// TIA Portal V17 export
// export: Created 2023-06-23T18:33:41.3605252Z, ExportSetting WithDefaults, DisplayName Totally Integrated Automation Portal, DisplayVersion V17, DisplayName TIA Portal Openness, DisplayVersion V17, DisplayName TIA Portal Version Control Interface, DisplayVersion V17, DisplayName STEP 7 Professional, DisplayVersion V17, DisplayName STEP 7 Safety, DisplayVersion V17, DisplayName WinCC Advanced / Unified PC, DisplayVersion V17
VAR_GLOBAL   // PLC tag table "28_ELR-3"
   "iELR-3" AT %I13.5 : Bool;
   "oELR-3" AT %Q13.0 : Bool;
END_VAR
